TYPE ACRMemoryDIntEvent EXTENDS ACRMemoryEvent :
STRUCT
	_Value : DINT;
END_STRUCT
END_TYPE

(* stored: Version 1.1.0.1, ProductVersion 3.1.4020.12
   DUT ACRMemoryDIntEvent: Id {e9c47628-8e63-423d-83e0-ebf954c1bba3} *)
